(********************* G.D S.p.A. - Technical Department ***********************************
This program has been generated automatically from Application Designer DE&F
********************************************************************************************)
PROGRAM dbg_csp_transfer_main_safety_drives_sd41300
VAR
  cha_smes_sis_shd : safety_integrated_series_shadow;
  chb_smes_sis_shd : safety_integrated_series_shadow;
END_VAR

_objects_manager();

IF	g_application_status <> APPLICATION_STATUS_RUNNING
THEN
	RETURN;
END_IF

CASE process_get_mode(CONVERSION_this := dbg_root.prc) OF
	MODE_ABSENT,
	MODE_INACTIVE:
		RETURN;
	MODE_TEST:
		RETURN;
END_CASE

ACTION _objects_manager:
IF	objects_initialization()
THEN
	safety_integrated_series_shadow_init(
		sim_mode:= SHADOW_SIMULATION_MODE_AUTOMATIC, 
		father:= csp_transfer_main_safety_drives_sd41300.cha_smes_sis, 
		process:= dbg_root.prc, 
		CONVERSION_this:= cha_smes_sis_shd);

	safety_integrated_series_shadow_init(
		sim_mode:= SHADOW_SIMULATION_MODE_AUTOMATIC, 
		father:= csp_transfer_main_safety_drives_sd41300.chb_smes_sis, 
		process:= dbg_root.prc, 
		CONVERSION_this:= chb_smes_sis_shd);

	RETURN;
END_IF

IF	objects_running()
THEN
	safety_integrated_series_shadow_cycle(cha_smes_sis_shd);
	safety_integrated_series_shadow_cycle(chb_smes_sis_shd);
END_IF
END_ACTION

END_PROGRAM

(* stored: Version 1.1.0.1, ProductVersion 3.1.4022.12
   POU dbg_csp_transfer_main_safety_drives_sd41300: Id {621076ce-363c-4687-b815-b0a039e76a50}, SpecialFunc None
   Action _objects_manager: Id {1f02fb7a-0a21-454a-97a6-148082b87de3} *)
